PROGRAM Move_Axis_Velocity
VAR
	fbMoveVelocity: MC_MoveVelocity;
	MoveVelocityExecute: BOOL;
	InVelocity: BOOL;
END_VAR

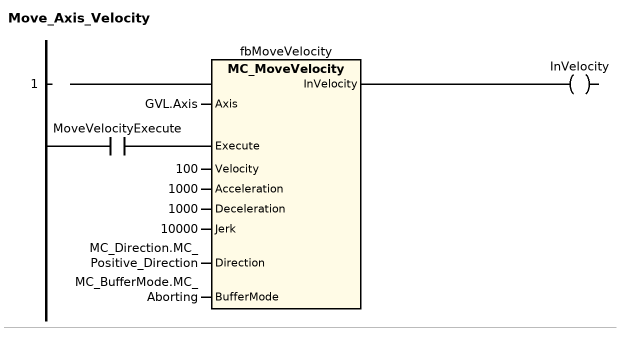
// NETWORK 1
fbMoveVelocity(
    Axis := GVL.Axis,
    Execute := MoveVelocityExecute,
    Velocity := 100,
    Acceleration := 1000,
    Deceleration := 1000,
    Jerk := 10000,
    Direction := MC_Direction.MC_Positive_Direction,
    BufferMode := MC_BufferMode.MC_Aborting); // MC_MoveVelocity
InVelocity := fbMoveVelocity.InVelocity;

END_PROGRAM

(* stored: Version 1.1.0.1, ProductVersion 3.1.4024.12
   POU Move_Axis_Velocity: Id {ce15da24-8d89-48a9-93b8-47af3bc89006}, SpecialFunc None *)
